PROGRAM MAIN
VAR	
	generateRecipe : BOOL;
	
	addRecipeToDB : AddRecipeToDatabase;
	validator : Validation;
	arrayHelpers : ArrayFunctions;
	
	resetAddRecipeToDatabase : AddRecipeToDatabase;
	resetValidation : Validation;
	resetArrayFunctions : ArrayFunctions;
	
	start : BOOL := TRUE;
END_VAR

validator(); //real time error/warning message generator

IF generateRecipe THEN
	addRecipeToDB();
	
	IF addRecipeToDB.finished THEN
		reset();
		//reset all variables
		generateRecipe := FALSE;
		RETURN;
	END_IF
END_IF

METHOD reset : BOOL
VAR_INPUT
END_VAR
//reset FBs
MEMCPY(ADR(addRecipeToDB), ADR(resetAddRecipeToDatabase), SIZEOF(AddRecipeToDatabase));
MEMCPY(ADR(validator), ADR(resetValidation), SIZEOF(Validation));
MEMCPY(ADR(arrayHelpers), ADR(resetArrayFunctions), SIZEOF(ArrayFunctions));

//reset fields
BundleData.id := '';
BundleData.weight := 0;
BundleData.length := 0;
BundleData.height := 0;
BundleData.width := 0;
BundleData.pieces := 0;
BundleData.piecesHeight := 0;
BundleData.piecesWidth := 0;
MEMSET(ADR(BundleData.requiredProcessing), 0, SIZEOF(BundleData.requiredProcessing));

ExtrusionData.extrusionWeight := 0;
ExtrusionData.extrusionHeight := 0;
ExtrusionData.extrusionWidth := 0;

MEMSET(ADR(StrapWrapRecipe.facePaper), 0, SIZEOF(StrapWrapRecipe.facePaper));
MEMSET(ADR(StrapWrapRecipe.faceCardboard), 0, SIZEOF(StrapWrapRecipe.faceCardboard));
MEMSET(ADR(StrapWrapRecipe.TopPaper), 0, SIZEOF(StrapWrapRecipe.TopPaper));
MEMSET(ADR(StrapWrapRecipe.SidesPaper), 0, SIZEOF(StrapWrapRecipe.SidesPaper));
MEMSET(ADR(StrapWrapRecipe.BottomPaper), 0, SIZEOF(StrapWrapRecipe.BottomPaper));
MEMSET(ADR(StrapWrapRecipe.Cardboard), 0, SIZEOF(StrapWrapRecipe.Cardboard));
MEMSET(ADR(StrapWrapRecipe.CornerGuard), 0, SIZEOF(StrapWrapRecipe.CornerGuard));
MEMSET(ADR(StrapWrapRecipe.Chipboard), 0, SIZEOF(StrapWrapRecipe.Chipboard));
MEMSET(ADR(StrapWrapRecipe.WoodBunk), 0, SIZEOF(StrapWrapRecipe.WoodBunk));
END_METHOD

END_PROGRAM

(* stored: Version 1.1.0.1, ProductVersion 3.1.4024.11
   POU MAIN: Id {37c506fa-13d3-435a-92ee-4c132e7c51fc}, SpecialFunc None
   Method reset: Id {0124509e-13da-40a2-aab9-bdaac9c2a94c} *)
